/// This struct contains variables that
/// * are read from outside (e.g. HMI) to retrieve information about the unit's current state and (temporary) parameters (= `publish`) 
/// * are written from outside (e.g. HMI) to control the unit via ADS (= `subscribe`) 
TYPE MoverCom :
STRUCT
  Publish : MoverComPublish;
  Subscribe : MoverComSubscribe;
END_STRUCT
END_TYPE

(* stored: Version 1.1.0.1
   DUT MoverCom: Id {0c48ed07-595e-40c7-893a-24344ed733f9} *)
